FUNCTION_BLOCK fb_flow_rate

VAR_INPUT
	// signal inputs
	ratio_in: REAL;
	xmeas_in: REAL;
	
	// parameters
	kc: REAL;
	ti: REAL;
	ts: REAL;
	hi: REAL := 100;
	lo: REAL;
	
	x0: REAL;
	
END_VAR

VAR_OUTPUT
	yout: REAL; // needs to be initialized by caller
END_VAR

VAR
	flow_rate_dpi: fb_discrete_pi := (kc := kc, ti := ti, ts := ts, hi := hi, lo := lo, x0:=x0);
END_VAR

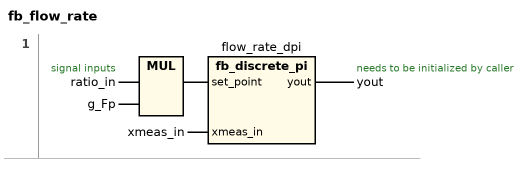
// NETWORK 1
//   ratio_in: signal inputs
//   yout: needs to be initialized by caller
flow_rate_dpi(set_point := ratio_in * g_Fp, xmeas_in := xmeas_in); // fb_discrete_pi
yout := flow_rate_dpi.yout;

END_FUNCTION_BLOCK

(* stored: Version 1.1.0.1, ProductVersion 3.1.0.26
   POU fb_flow_rate: Id {e3a0ade3-b22e-4736-b804-c9e196e4ed5c} *)
